// TIA Portal V17 export
// export: Created 2025-05-22T12:26:37.545947Z, ExportSetting WithDefaults, DisplayName Totally Integrated Automation Portal, DisplayVersion V17 Update 8, DisplayName TIA Portal Openness, DisplayVersion V17 Update 8, DisplayName TIA Portal Version Control Interface, DisplayVersion V17, DisplayName SINAMICS Startdrive Advanced, DisplayVersion V17 SP2, DisplayName SINAMICS Startdrive G110M, G120, G120C, G120D, G120P, G115D, DisplayVersion V17 SP2, DisplayName SINAMICS Startdrive G130, G150, S120, S150, SINAMICS MV, S210, DisplayVersion V17 SP2, DisplayName STEP 7 Professional, DisplayVersion V17 Update 8, DisplayName SINUMERIK ONE STEP 7 Toolbox, DisplayVersion V17 Update 12, DisplayName SINUMERIK ONE PLC Basic Program Plus, DisplayVersion V17 Update 12, DisplayName SINUMERIK 840D sl STEP 7 Toolbox, DisplayVersion V17 Update 12, DisplayName STEP 7 Safety, DisplayVersion V17 Update 6, DisplayName WinCC Advanced, DisplayVersion V17 Update 8
FUNCTION_BLOCK "FB1502_PROTECTION_GAS_VALVE"   // FB1502, LAD
{ S7_Optimized_Access := 'FALSE' }
VERSION : 0.1
// stored: AutoNumber false, IsIECCheckEnabled false, SetENOAutomatically false, UDAEnableTagReadback false
   VAR_INPUT
      FLOW_INPUT : Real;   // FLOW INPUT
      TEMPERATURE_INPUT : Real;   // TEMPERATURE INPUT
      LASER_READY_INPUT : Bool;   // LASER READY INPUT
      SWITCH_ON_CONDITIONS : Bool;   // SWITCH ON CONDITIONS
      SWITCH_OFF_CONDITIONS : Bool;   // SWITCH OFF CONDITIONS
      HMI_LINE_REQUEST : Bool;   // HMI LINE REQUEST
      SWITCH_ON_AUTO_REQUEST : Bool;   // AUTO SWITCH ON REQUEST
      SWITCH_OFF_AUTO_REQUEST : Bool;   // AUTO SWITCH OFF REQUEST
      SWITCH_OFF_GLOBAL_REQUEST : Bool;   // SWITCH OFF GLOBAL REQUEST (AUTO/SEMI/MAN)
      POWDER_ENABLED : Bool;
      UNIT_ALARM : UInt;   // UNIT NUMBER MIN. NUMBER=1 MAX. NUMBER=4
      STATION_ALARM : UInt;   // STATION NUMBER MIN. NUMBER=0 MAX. NUMBER=4
   END_VAR
   VAR_OUTPUT
      SWITCHED_ON : Bool;   // SWITCHED ON
      SWITCHED_OFF : Bool;   // SWITCHED OFF
      SIMULTANEITY_ALARM : Bool;   // SIMULTANEITY ALARM
      TIME_EXCEEDED_ALARM : Bool;   // TIME EXCEEDED ALARM
      SWITCH_ON_ALARM : Bool;   // SWITCH ON ALARM
      SWITCH_OFF_ALARM : Bool;   // SWITCH OFF ALARM
      GAS_FLOW_LOW_WARNING : Bool;   // GAS FLOW LOW WARNING
      GAS_FLOW_LOW_ALARM : Bool;   // GAS FLOW LOW ALARM
      GAS_FLOW_HIGH_WARNING : Bool;   // GAS FLOW HIGH WARNING
      GAS_FLOW_HIGH_ALARM : Bool;   // GAS FLOW HIGH ALARM
      GAS_TEMP_LOW_WARNING : Bool;   // GAS TEMPERATURE LOW WARNING
      GAS_TEMP_LOW_ALARM : Bool;   // GAS TEMPERATURE LOW ALARM
      GAS_TEMP_HIGH_WARNING : Bool;   // GAS TEMPERATURE HIGH WARNING
      GAS_TEMP_HIGH_ALARM : Bool;   // GAS TEMPERATURE HIGH ALARM
      ANY_ALARM_PRESENT : Bool;   // ANY ALARM PRESENT
      HMI_MOTION_EXECUTABILITY_LEFT : Bool;   // HMI MOTION EXECUTABILITY LEFT
      HMI_MOTION_EXECUTABILITY_RIGHT : Bool;   // HMI MOTION EXECUTABILITY RIGHT
      HMI_MOTION_END_POS_LEFT : Bool;   // HMI MOTION END POSITION LEFT
      HMI_MOTION_END_POS_RIGHT : Bool;   // HMI MOTION END POSITION RIGHT
      HMI_MOTION_ACTIVE_LEFT : Bool;   // HMI MOTION ACTIVE LEFT
      HMI_MOTION_ACTIVE_RIGHT : Bool;   // HMI MOTION ACTIVE RIGHT
      GAS_FLOW_SETPOINT : Real;   // GAS FLOW SETPOINT
      SWITCH_ON : Bool;   // SWITCH ON OUTPUT
      SWITCH_OFF : Bool;   // SWITCH OFF OUTPUT
   END_VAR
   VAR DB_SPECIFIC
      VALVE { S7_SetPoint := 'True'} : "ASPIRATION";
      HMI_VARIBLES : Struct
         HMI_GAS_FLOW_SETPOINT { S7_SetPoint := 'True'} : Real;
         GAS_FLOW_LOW_WARNING_VALUE : Real;
         GAS_FLOW_LOW_ALARM_VALUE : Real;
         GAS_FLOW_HIGH_WARNING_VALUE : Real;
         GAS_FLOW_HIGH_ALARM_VALUE : Real;
         TEMP_LOW_WARNING_VALUE : Real;
         TEMP_LOW_ALARM_VALUE : Real;
         TEMP_HIGH_WARNING_VALUE : Real;
         TEMP_HIGH_ALARM_VALUE : Real;
      END_STRUCT;
      FLOW_VALUE : Real;
      AUX_TEMP { S7_SetPoint := 'True'} : Real;   // AUX TEMPERATURE
      TEMPERATURE_VALUE { S7_SetPoint := 'True'} : Real;   // TEMPERATURE VALUE
      TIMER_SWITCHED_ON { S7_SetPoint := 'True'} : TON_TIME;   // SWITCHED ON TIMER
      TIMER_SWITCHED_OFF { S7_SetPoint := 'True'} : TON_TIME;   // SWITCHED OFF TIMER
      TIMER_SIMULTANEITY { S7_SetPoint := 'True'} : TON_TIME;   // SIMULTANEITY TIMER
      TIMER_TIME_EXCEEDED { S7_SetPoint := 'True'} : TON_TIME;   // TIME EXCEEDED TIMER
      GAS_FLOW_LOW_WARNING_DELAY { S7_SetPoint := 'True'} : TON_TIME;
      GAS_FLOW_LOW_ALARM_DELAY { S7_SetPoint := 'True'} : TON_TIME;
      PULSE { S7_SetPoint := 'True'} : Bool;
   END_VAR
   VAR_TEMP
      DB_NUMBER : DInt;   // DB NUMBER FOR ALARM AND HELP DECODING
   END_VAR
   // TIMER_SWITCHED_ON.PT := T#100MS;
   // TIMER_SWITCHED_OFF.PT := T#300MS;
   // TIMER_SIMULTANEITY.PT := T#100MS;
   // TIMER_TIME_EXCEEDED.PT := T#2S;
   VAR_TEMP   // added for the SCL form of the ladder/FBD networks
      _w1 : Bool;
      _w2 : Bool;
   END_VAR
BEGIN

NETWORK
TITLE = READ INSTANCE DB
      L     DINO;
      +     10#800000;
      T     #DB_NUMBER;


REGION Network 2: INPUT
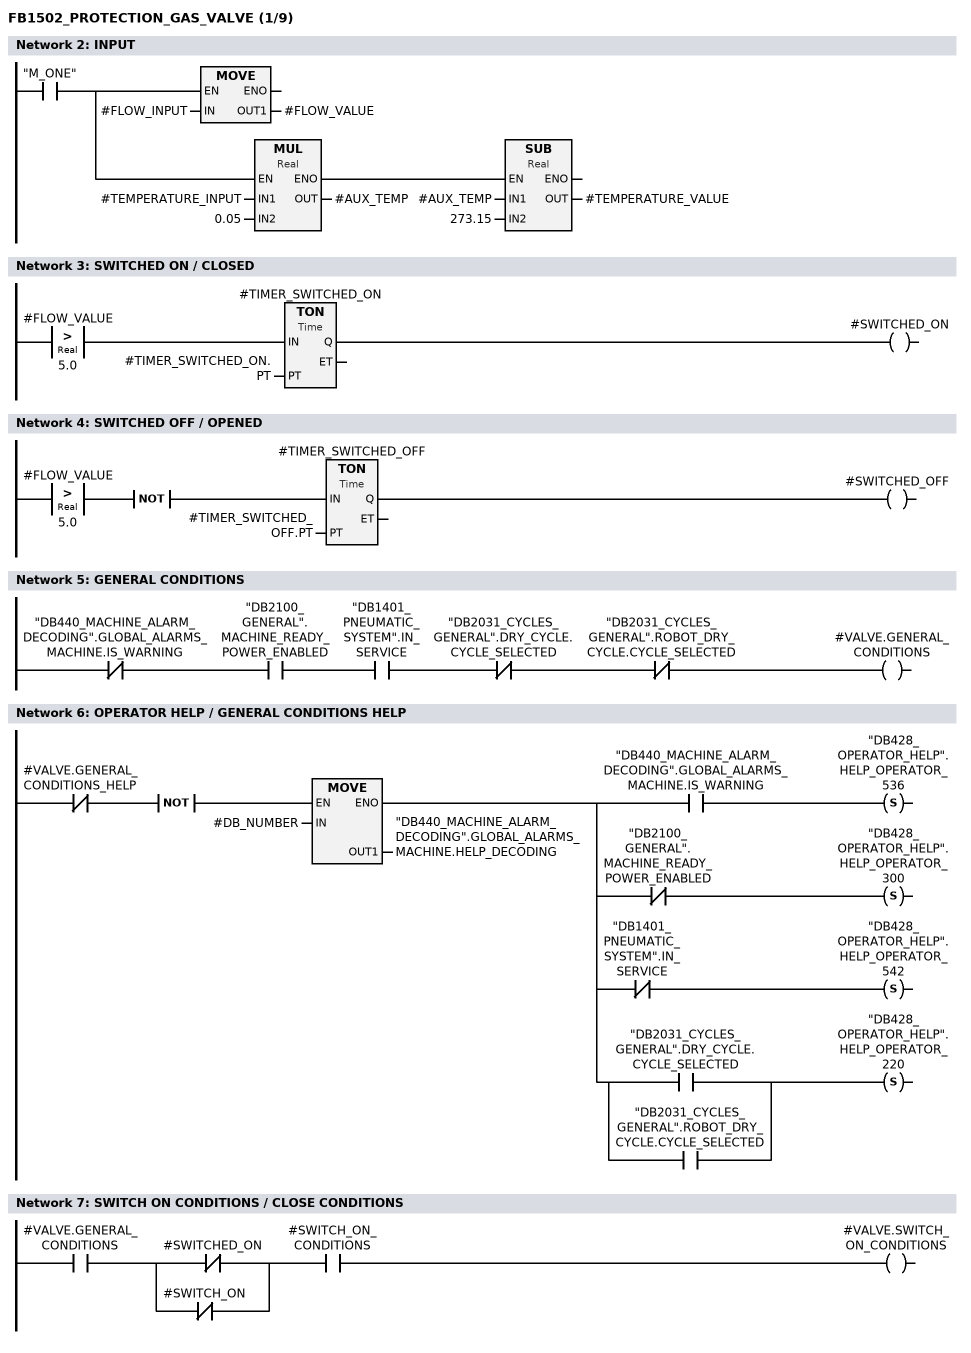
   RUNG wire#powerrail
      Contact( "M_ONE" )
      wire#w1
      Move(in := #FLOW_INPUT, out1 => #FLOW_VALUE)
   END_RUNG
   RUNG wire#w1
      { S7_Templates := "SrcType := Real" } Mul(in1 := #TEMPERATURE_INPUT, in2 := 0.05, out => #AUX_TEMP)
      { S7_Templates := "SrcType := Real" } Sub(in1 := #AUX_TEMP, in2 := 273.15, out => #TEMPERATURE_VALUE)
   END_RUNG
   // the same network as SCL:
   IF "M_ONE" THEN
       #FLOW_VALUE := #FLOW_INPUT;
       #AUX_TEMP := #TEMPERATURE_INPUT * 0.05;
       #TEMPERATURE_VALUE := #AUX_TEMP - 273.15;
   END_IF;
END_REGION

REGION Network 3: SWITCHED ON / CLOSED
   RUNG wire#powerrail
      { S7_Templates := "SrcType := Real" } GT_Contact(in1 := #FLOW_VALUE, in2 := 5.0)
      { S7_Templates := "time_type := Time" } #TIMER_SWITCHED_ON.TON(pt := #TIMER_SWITCHED_ON.PT, et =>)
      Coil( #SWITCHED_ON )
   END_RUNG
   // the same network as SCL:
   #TIMER_SWITCHED_ON(IN := #FLOW_VALUE > 5.0, PT := #TIMER_SWITCHED_ON.PT);   // TON
   #SWITCHED_ON := #TIMER_SWITCHED_ON.Q;
END_REGION

REGION Network 4: SWITCHED OFF / OPENED
   RUNG wire#powerrail
      { S7_Templates := "SrcType := Real" } GT_Contact(in1 := #FLOW_VALUE, in2 := 5.0)
      Not()
      { S7_Templates := "time_type := Time" } #TIMER_SWITCHED_OFF.TON(pt := #TIMER_SWITCHED_OFF.PT, et =>)
      Coil( #SWITCHED_OFF )
   END_RUNG
   // the same network as SCL:
   #TIMER_SWITCHED_OFF(IN := NOT (#FLOW_VALUE > 5.0), PT := #TIMER_SWITCHED_OFF.PT);   // TON
   #SWITCHED_OFF := #TIMER_SWITCHED_OFF.Q;
END_REGION

REGION Network 5: GENERAL CONDITIONS
   RUNG wire#powerrail
      I_Contact( "DB440_MACHINE_ALARM_DECODING".GLOBAL_ALARMS_MACHINE.IS_WARNING )
      Contact( "DB2100_GENERAL".MACHINE_READY_POWER_ENABLED )
      Contact( "DB1401_PNEUMATIC_SYSTEM".IN_SERVICE )
      I_Contact( "DB2031_CYCLES_GENERAL".DRY_CYCLE.CYCLE_SELECTED )
      I_Contact( "DB2031_CYCLES_GENERAL".ROBOT_DRY_CYCLE.CYCLE_SELECTED )
      Coil( #VALVE.GENERAL_CONDITIONS )
   END_RUNG
   // the same network as SCL:
   #VALVE.GENERAL_CONDITIONS := NOT "DB440_MACHINE_ALARM_DECODING".GLOBAL_ALARMS_MACHINE.IS_WARNING AND "DB2100_GENERAL".MACHINE_READY_POWER_ENABLED AND "DB1401_PNEUMATIC_SYSTEM".IN_SERVICE AND NOT "DB2031_CYCLES_GENERAL".DRY_CYCLE.CYCLE_SELECTED AND NOT "DB2031_CYCLES_GENERAL".ROBOT_DRY_CYCLE.CYCLE_SELECTED;
END_REGION

REGION Network 6: OPERATOR HELP / GENERAL CONDITIONS HELP
   RUNG wire#powerrail
      I_Contact( #VALVE.GENERAL_CONDITIONS_HELP )
      Not()
      { S7_GenerateENO := "TRUE" } Move(in := #DB_NUMBER, out1 => "DB440_MACHINE_ALARM_DECODING".GLOBAL_ALARMS_MACHINE.HELP_DECODING)
      wire#w1
      Contact( "DB440_MACHINE_ALARM_DECODING".GLOBAL_ALARMS_MACHINE.IS_WARNING )
      S_Coil( "DB428_OPERATOR_HELP".HELP_OPERATOR_536 )
   END_RUNG
   RUNG wire#w1
      I_Contact( "DB2100_GENERAL".MACHINE_READY_POWER_ENABLED )
      S_Coil( "DB428_OPERATOR_HELP".HELP_OPERATOR_300 )
   END_RUNG
   RUNG wire#w1
      I_Contact( "DB1401_PNEUMATIC_SYSTEM".IN_SERVICE )
      S_Coil( "DB428_OPERATOR_HELP".HELP_OPERATOR_542 )
   END_RUNG
   RUNG wire#w1
      Contact( "DB2031_CYCLES_GENERAL".DRY_CYCLE.CYCLE_SELECTED )
      wire#w2
      S_Coil( "DB428_OPERATOR_HELP".HELP_OPERATOR_220 )
   END_RUNG
   RUNG wire#w1
      Contact( "DB2031_CYCLES_GENERAL".ROBOT_DRY_CYCLE.CYCLE_SELECTED )
   END_RUNG wire#w2
   // the same network as SCL:
   // ENO of a box is taken as its EN; it also drops when the box reports an error
   #_w1 := NOT (NOT #VALVE.GENERAL_CONDITIONS_HELP);
   IF #_w1 THEN "DB440_MACHINE_ALARM_DECODING".GLOBAL_ALARMS_MACHINE.HELP_DECODING := #DB_NUMBER; END_IF;
   IF #_w1 AND "DB440_MACHINE_ALARM_DECODING".GLOBAL_ALARMS_MACHINE.IS_WARNING THEN
       "DB428_OPERATOR_HELP".HELP_OPERATOR_536 := TRUE;
   END_IF;
   IF #_w1 AND NOT "DB2100_GENERAL".MACHINE_READY_POWER_ENABLED THEN
       "DB428_OPERATOR_HELP".HELP_OPERATOR_300 := TRUE;
   END_IF;
   IF #_w1 AND NOT "DB1401_PNEUMATIC_SYSTEM".IN_SERVICE THEN
       "DB428_OPERATOR_HELP".HELP_OPERATOR_542 := TRUE;
   END_IF;
   IF #_w1 AND ("DB2031_CYCLES_GENERAL".DRY_CYCLE.CYCLE_SELECTED OR "DB2031_CYCLES_GENERAL".ROBOT_DRY_CYCLE.CYCLE_SELECTED) THEN
       "DB428_OPERATOR_HELP".HELP_OPERATOR_220 := TRUE;
   END_IF;
END_REGION

REGION Network 7: SWITCH ON CONDITIONS / CLOSE CONDITIONS
   RUNG wire#powerrail
      Contact( #VALVE.GENERAL_CONDITIONS )
      wire#w1
      I_Contact( #SWITCHED_ON )
      wire#w2
      Contact( #SWITCH_ON_CONDITIONS )
      Coil( #VALVE.SWITCH_ON_CONDITIONS )
   END_RUNG
   RUNG wire#w1
      I_Contact( #SWITCH_ON )
   END_RUNG wire#w2
   // the same network as SCL:
   #VALVE.SWITCH_ON_CONDITIONS := #VALVE.GENERAL_CONDITIONS AND (NOT #SWITCHED_ON OR NOT #SWITCH_ON) AND #SWITCH_ON_CONDITIONS;
END_REGION

REGION Network 8: OPERATOR HELP / CLOSE CONDITIONS HELP
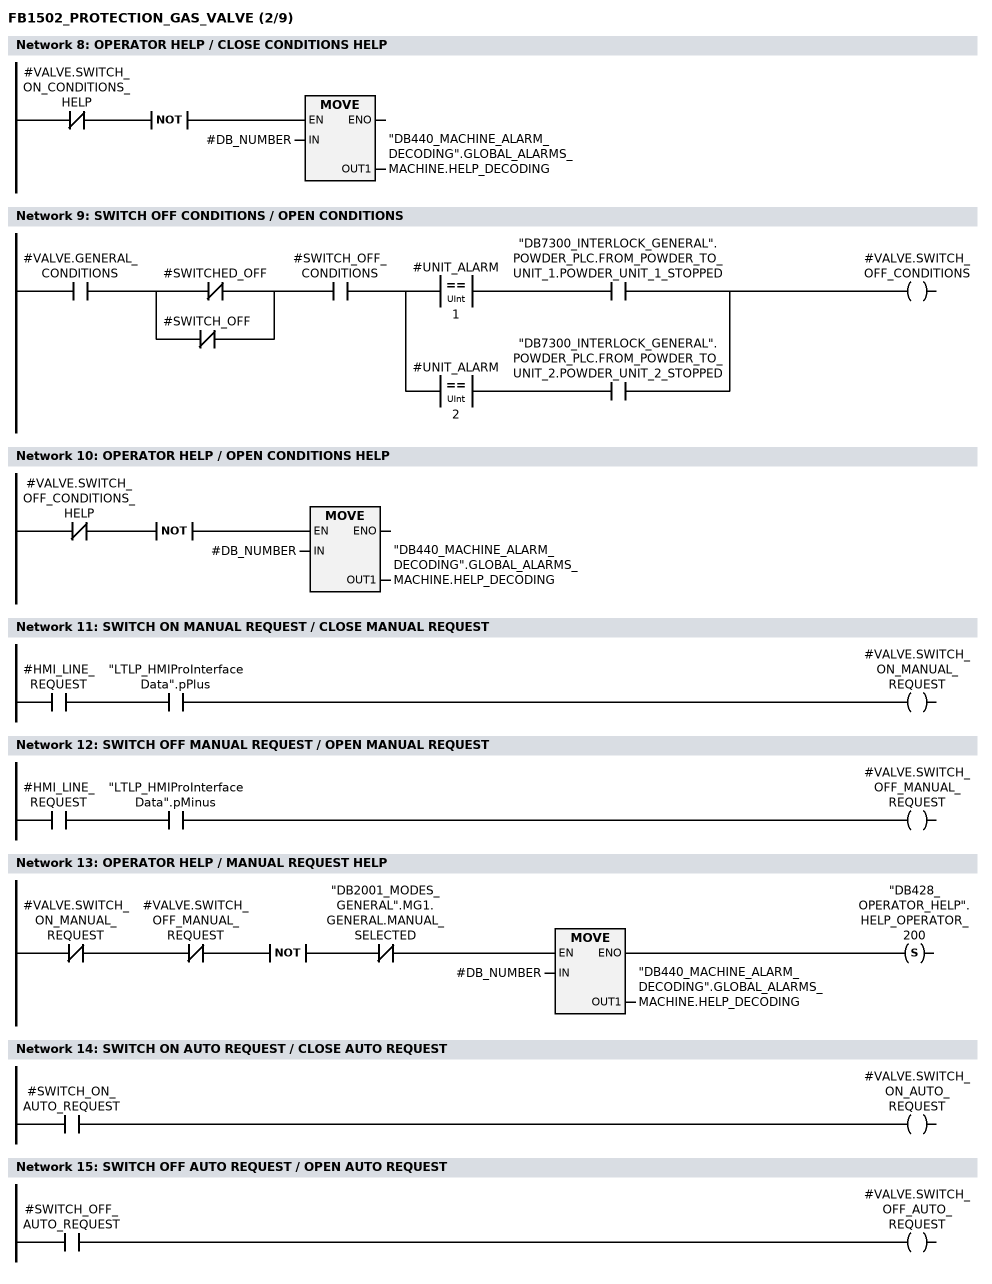
   RUNG wire#powerrail
      I_Contact( #VALVE.SWITCH_ON_CONDITIONS_HELP )
      Not()
      { S7_GenerateENO := "TRUE" } Move(in := #DB_NUMBER, out1 => "DB440_MACHINE_ALARM_DECODING".GLOBAL_ALARMS_MACHINE.HELP_DECODING)
   END_RUNG
   // the same network as SCL:
   IF NOT (NOT #VALVE.SWITCH_ON_CONDITIONS_HELP) THEN
       "DB440_MACHINE_ALARM_DECODING".GLOBAL_ALARMS_MACHINE.HELP_DECODING := #DB_NUMBER;
   END_IF;
END_REGION

REGION Network 9: SWITCH OFF CONDITIONS / OPEN CONDITIONS
   RUNG wire#powerrail
      Contact( #VALVE.GENERAL_CONDITIONS )
      wire#w1
      I_Contact( #SWITCHED_OFF )
      wire#w2
      Contact( #SWITCH_OFF_CONDITIONS )
      wire#w3
      { S7_Templates := "SrcType := UInt" } EQ_Contact(in1 := #UNIT_ALARM, in2 := 1)
      Contact( "DB7300_INTERLOCK_GENERAL".POWDER_PLC.FROM_POWDER_TO_UNIT_1.POWDER_UNIT_1_STOPPED )
      wire#w4
      Coil( #VALVE.SWITCH_OFF_CONDITIONS )
   END_RUNG
   RUNG wire#w1
      I_Contact( #SWITCH_OFF )
   END_RUNG wire#w2
   RUNG wire#w3
      { S7_Templates := "SrcType := UInt" } EQ_Contact(in1 := #UNIT_ALARM, in2 := 2)
      Contact( "DB7300_INTERLOCK_GENERAL".POWDER_PLC.FROM_POWDER_TO_UNIT_2.POWDER_UNIT_2_STOPPED )
   END_RUNG wire#w4
   // the same network as SCL:
   #VALVE.SWITCH_OFF_CONDITIONS := #VALVE.GENERAL_CONDITIONS AND (NOT #SWITCHED_OFF OR NOT #SWITCH_OFF) AND #SWITCH_OFF_CONDITIONS AND (((#UNIT_ALARM = 1) AND "DB7300_INTERLOCK_GENERAL".POWDER_PLC.FROM_POWDER_TO_UNIT_1.POWDER_UNIT_1_STOPPED) OR ((#UNIT_ALARM = 2) AND "DB7300_INTERLOCK_GENERAL".POWDER_PLC.FROM_POWDER_TO_UNIT_2.POWDER_UNIT_2_STOPPED));
END_REGION

REGION Network 10: OPERATOR HELP / OPEN CONDITIONS HELP
   RUNG wire#powerrail
      I_Contact( #VALVE.SWITCH_OFF_CONDITIONS_HELP )
      Not()
      { S7_GenerateENO := "TRUE" } Move(in := #DB_NUMBER, out1 => "DB440_MACHINE_ALARM_DECODING".GLOBAL_ALARMS_MACHINE.HELP_DECODING)
   END_RUNG
   // the same network as SCL:
   IF NOT (NOT #VALVE.SWITCH_OFF_CONDITIONS_HELP) THEN
       "DB440_MACHINE_ALARM_DECODING".GLOBAL_ALARMS_MACHINE.HELP_DECODING := #DB_NUMBER;
   END_IF;
END_REGION

REGION Network 11: SWITCH ON MANUAL REQUEST / CLOSE MANUAL REQUEST
   RUNG wire#powerrail
      Contact( #HMI_LINE_REQUEST )
      Contact( "LTLP_HMIProInterfaceData".pPlus )
      Coil( #VALVE.SWITCH_ON_MANUAL_REQUEST )
   END_RUNG
   // the same network as SCL:
   #VALVE.SWITCH_ON_MANUAL_REQUEST := #HMI_LINE_REQUEST AND "LTLP_HMIProInterfaceData".pPlus;
END_REGION

REGION Network 12: SWITCH OFF MANUAL REQUEST / OPEN MANUAL REQUEST
   RUNG wire#powerrail
      Contact( #HMI_LINE_REQUEST )
      Contact( "LTLP_HMIProInterfaceData".pMinus )
      Coil( #VALVE.SWITCH_OFF_MANUAL_REQUEST )
   END_RUNG
   // the same network as SCL:
   #VALVE.SWITCH_OFF_MANUAL_REQUEST := #HMI_LINE_REQUEST AND "LTLP_HMIProInterfaceData".pMinus;
END_REGION

REGION Network 13: OPERATOR HELP / MANUAL REQUEST HELP
   RUNG wire#powerrail
      I_Contact( #VALVE.SWITCH_ON_MANUAL_REQUEST )
      I_Contact( #VALVE.SWITCH_OFF_MANUAL_REQUEST )
      Not()
      I_Contact( "DB2001_MODES_GENERAL".MG1.GENERAL.MANUAL_SELECTED )
      { S7_GenerateENO := "TRUE" } Move(in := #DB_NUMBER, out1 => "DB440_MACHINE_ALARM_DECODING".GLOBAL_ALARMS_MACHINE.HELP_DECODING)
      S_Coil( "DB428_OPERATOR_HELP".HELP_OPERATOR_200 )
   END_RUNG
   // the same network as SCL:
   // ENO of a box is taken as its EN; it also drops when the box reports an error
   IF NOT (NOT #VALVE.SWITCH_ON_MANUAL_REQUEST AND NOT #VALVE.SWITCH_OFF_MANUAL_REQUEST) AND NOT "DB2001_MODES_GENERAL".MG1.GENERAL.MANUAL_SELECTED THEN
       "DB440_MACHINE_ALARM_DECODING".GLOBAL_ALARMS_MACHINE.HELP_DECODING := #DB_NUMBER;
       "DB428_OPERATOR_HELP".HELP_OPERATOR_200 := TRUE;
   END_IF;
END_REGION

REGION Network 14: SWITCH ON AUTO REQUEST / CLOSE AUTO REQUEST
   RUNG wire#powerrail
      Contact( #SWITCH_ON_AUTO_REQUEST )
      Coil( #VALVE.SWITCH_ON_AUTO_REQUEST )
   END_RUNG
   // the same network as SCL:
   #VALVE.SWITCH_ON_AUTO_REQUEST := #SWITCH_ON_AUTO_REQUEST;
END_REGION

REGION Network 15: SWITCH OFF AUTO REQUEST / OPEN AUTO REQUEST
   RUNG wire#powerrail
      Contact( #SWITCH_OFF_AUTO_REQUEST )
      Coil( #VALVE.SWITCH_OFF_AUTO_REQUEST )
   END_RUNG
   // the same network as SCL:
   #VALVE.SWITCH_OFF_AUTO_REQUEST := #SWITCH_OFF_AUTO_REQUEST;
END_REGION

REGION Network 16: SWITCH ON GLOBAL REQUEST / CLOSE GLOBAL REQUEST
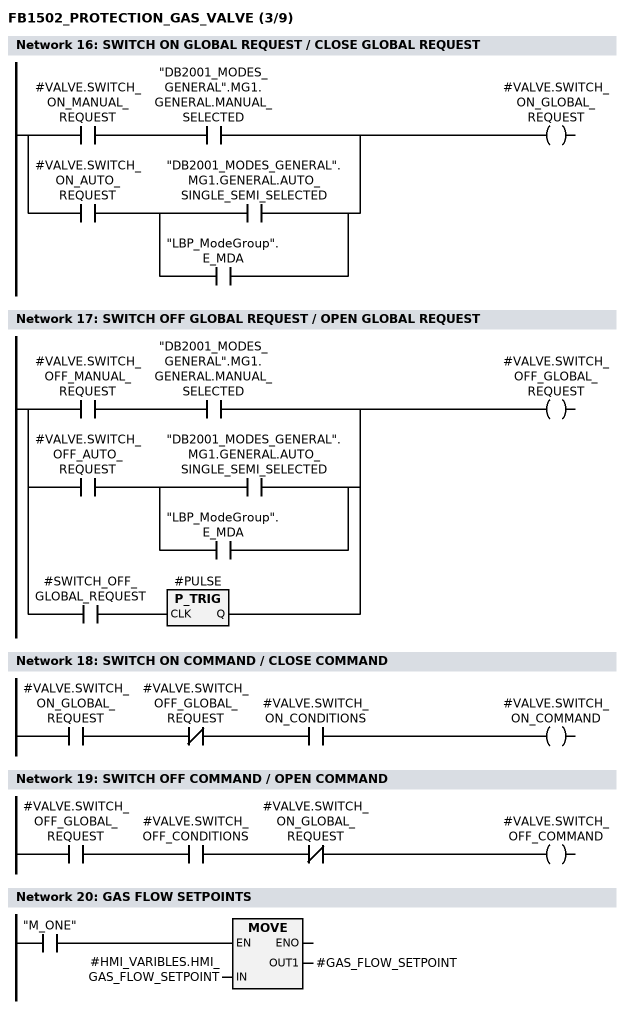
   RUNG wire#powerrail
      Contact( #VALVE.SWITCH_ON_MANUAL_REQUEST )
      Contact( "DB2001_MODES_GENERAL".MG1.GENERAL.MANUAL_SELECTED )
      wire#w1
      Coil( #VALVE.SWITCH_ON_GLOBAL_REQUEST )
   END_RUNG
   RUNG wire#powerrail
      Contact( #VALVE.SWITCH_ON_AUTO_REQUEST )
      wire#w2
      Contact( "DB2001_MODES_GENERAL".MG1.GENERAL.AUTO_SINGLE_SEMI_SELECTED )
   END_RUNG wire#w1
   RUNG wire#w2
      Contact( "LBP_ModeGroup".E_MDA )
   END_RUNG wire#w1
   // the same network as SCL:
   #VALVE.SWITCH_ON_GLOBAL_REQUEST := (#VALVE.SWITCH_ON_MANUAL_REQUEST AND "DB2001_MODES_GENERAL".MG1.GENERAL.MANUAL_SELECTED) OR (#VALVE.SWITCH_ON_AUTO_REQUEST AND ("DB2001_MODES_GENERAL".MG1.GENERAL.AUTO_SINGLE_SEMI_SELECTED OR "LBP_ModeGroup".E_MDA));
END_REGION

REGION Network 17: SWITCH OFF GLOBAL REQUEST / OPEN GLOBAL REQUEST
   RUNG wire#powerrail
      Contact( #VALVE.SWITCH_OFF_MANUAL_REQUEST )
      Contact( "DB2001_MODES_GENERAL".MG1.GENERAL.MANUAL_SELECTED )
      wire#w1
      Coil( #VALVE.SWITCH_OFF_GLOBAL_REQUEST )
   END_RUNG
   RUNG wire#powerrail
      Contact( #VALVE.SWITCH_OFF_AUTO_REQUEST )
      wire#w2
      Contact( "DB2001_MODES_GENERAL".MG1.GENERAL.AUTO_SINGLE_SEMI_SELECTED )
   END_RUNG wire#w1
   RUNG wire#w2
      Contact( "LBP_ModeGroup".E_MDA )
   END_RUNG wire#w1
   RUNG wire#powerrail
      Contact( #SWITCH_OFF_GLOBAL_REQUEST )
      P_Trig( #PULSE )
   END_RUNG wire#w1
   // the same network as SCL:
   #_w1 := #SWITCH_OFF_GLOBAL_REQUEST AND NOT #PULSE;   // rising edge
   #PULSE := #SWITCH_OFF_GLOBAL_REQUEST;
   #VALVE.SWITCH_OFF_GLOBAL_REQUEST := (#VALVE.SWITCH_OFF_MANUAL_REQUEST AND "DB2001_MODES_GENERAL".MG1.GENERAL.MANUAL_SELECTED) OR (#VALVE.SWITCH_OFF_AUTO_REQUEST AND ("DB2001_MODES_GENERAL".MG1.GENERAL.AUTO_SINGLE_SEMI_SELECTED OR "LBP_ModeGroup".E_MDA)) OR #_w1;
END_REGION

REGION Network 18: SWITCH ON COMMAND / CLOSE COMMAND
   RUNG wire#powerrail
      Contact( #VALVE.SWITCH_ON_GLOBAL_REQUEST )
      I_Contact( #VALVE.SWITCH_OFF_GLOBAL_REQUEST )
      Contact( #VALVE.SWITCH_ON_CONDITIONS )
      Coil( #VALVE.SWITCH_ON_COMMAND )
   END_RUNG
   // the same network as SCL:
   #VALVE.SWITCH_ON_COMMAND := #VALVE.SWITCH_ON_GLOBAL_REQUEST AND NOT #VALVE.SWITCH_OFF_GLOBAL_REQUEST AND #VALVE.SWITCH_ON_CONDITIONS;
END_REGION

REGION Network 19: SWITCH OFF COMMAND / OPEN COMMAND
   RUNG wire#powerrail
      Contact( #VALVE.SWITCH_OFF_GLOBAL_REQUEST )
      Contact( #VALVE.SWITCH_OFF_CONDITIONS )
      I_Contact( #VALVE.SWITCH_ON_GLOBAL_REQUEST )
      Coil( #VALVE.SWITCH_OFF_COMMAND )
   END_RUNG
   // the same network as SCL:
   #VALVE.SWITCH_OFF_COMMAND := #VALVE.SWITCH_OFF_GLOBAL_REQUEST AND #VALVE.SWITCH_OFF_CONDITIONS AND NOT #VALVE.SWITCH_ON_GLOBAL_REQUEST;
END_REGION

REGION Network 20: GAS FLOW SETPOINTS
   RUNG wire#powerrail
      Contact( "M_ONE" )
      Move(in := #HMI_VARIBLES.HMI_GAS_FLOW_SETPOINT, out1 => #GAS_FLOW_SETPOINT)
   END_RUNG
   // the same network as SCL:
   IF "M_ONE" THEN #GAS_FLOW_SETPOINT := #HMI_VARIBLES.HMI_GAS_FLOW_SETPOINT; END_IF;
END_REGION

REGION Network 21: SWITCH ON OUTPUT / CLOSE
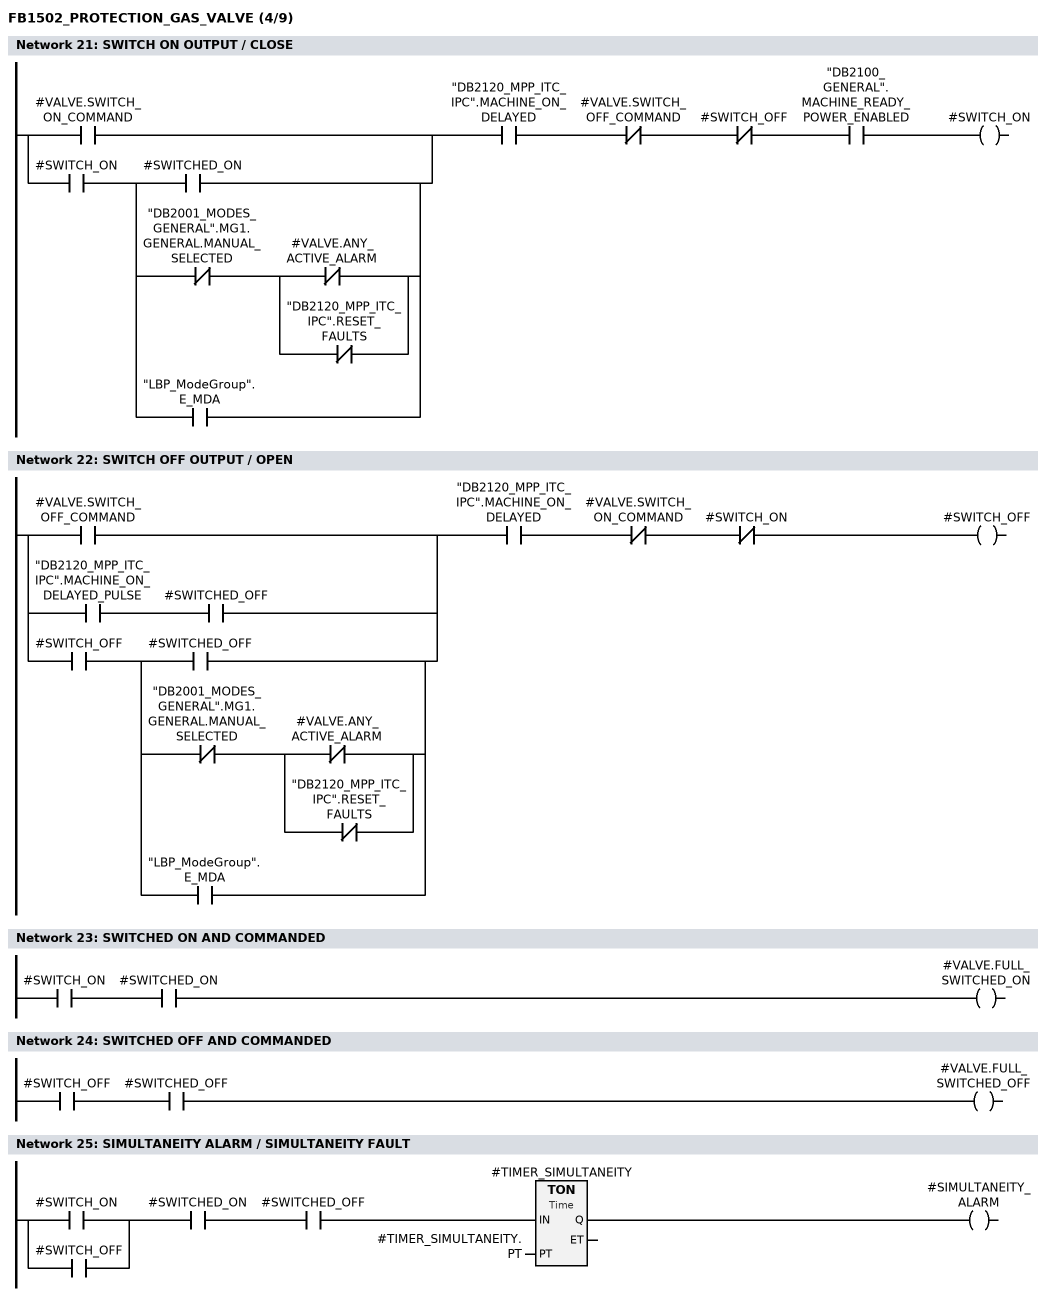
   RUNG wire#powerrail
      Contact( #VALVE.SWITCH_ON_COMMAND )
      wire#w1
      Contact( "DB2120_MPP_ITC_IPC".MACHINE_ON_DELAYED )
      I_Contact( #VALVE.SWITCH_OFF_COMMAND )
      I_Contact( #SWITCH_OFF )
      Contact( "DB2100_GENERAL".MACHINE_READY_POWER_ENABLED )
      Coil( #SWITCH_ON )
   END_RUNG
   RUNG wire#powerrail
      Contact( #SWITCH_ON )
      wire#w2
      Contact( #SWITCHED_ON )
   END_RUNG wire#w1
   RUNG wire#w2
      I_Contact( "DB2001_MODES_GENERAL".MG1.GENERAL.MANUAL_SELECTED )
      wire#w3
      I_Contact( #VALVE.ANY_ACTIVE_ALARM )
   END_RUNG wire#w1
   RUNG wire#w3
      I_Contact( "DB2120_MPP_ITC_IPC".RESET_FAULTS )
   END_RUNG wire#w1
   RUNG wire#w2
      Contact( "LBP_ModeGroup".E_MDA )
   END_RUNG wire#w1
   // the same network as SCL:
   #SWITCH_ON := (#VALVE.SWITCH_ON_COMMAND OR (#SWITCH_ON AND (#SWITCHED_ON OR (NOT "DB2001_MODES_GENERAL".MG1.GENERAL.MANUAL_SELECTED AND (NOT #VALVE.ANY_ACTIVE_ALARM OR NOT "DB2120_MPP_ITC_IPC".RESET_FAULTS)) OR "LBP_ModeGroup".E_MDA))) AND "DB2120_MPP_ITC_IPC".MACHINE_ON_DELAYED AND NOT #VALVE.SWITCH_OFF_COMMAND AND NOT #SWITCH_OFF AND "DB2100_GENERAL".MACHINE_READY_POWER_ENABLED;
END_REGION

REGION Network 22: SWITCH OFF OUTPUT / OPEN
   RUNG wire#powerrail
      Contact( #VALVE.SWITCH_OFF_COMMAND )
      wire#w1
      Contact( "DB2120_MPP_ITC_IPC".MACHINE_ON_DELAYED )
      I_Contact( #VALVE.SWITCH_ON_COMMAND )
      I_Contact( #SWITCH_ON )
      Coil( #SWITCH_OFF )
   END_RUNG
   RUNG wire#powerrail
      Contact( "DB2120_MPP_ITC_IPC".MACHINE_ON_DELAYED_PULSE )
      Contact( #SWITCHED_OFF )
   END_RUNG wire#w1
   RUNG wire#powerrail
      Contact( #SWITCH_OFF )
      wire#w2
      Contact( #SWITCHED_OFF )
   END_RUNG wire#w1
   RUNG wire#w2
      I_Contact( "DB2001_MODES_GENERAL".MG1.GENERAL.MANUAL_SELECTED )
      wire#w3
      I_Contact( #VALVE.ANY_ACTIVE_ALARM )
   END_RUNG wire#w1
   RUNG wire#w3
      I_Contact( "DB2120_MPP_ITC_IPC".RESET_FAULTS )
   END_RUNG wire#w1
   RUNG wire#w2
      Contact( "LBP_ModeGroup".E_MDA )
   END_RUNG wire#w1
   // the same network as SCL:
   #SWITCH_OFF := (#VALVE.SWITCH_OFF_COMMAND OR ("DB2120_MPP_ITC_IPC".MACHINE_ON_DELAYED_PULSE AND #SWITCHED_OFF) OR (#SWITCH_OFF AND (#SWITCHED_OFF OR (NOT "DB2001_MODES_GENERAL".MG1.GENERAL.MANUAL_SELECTED AND (NOT #VALVE.ANY_ACTIVE_ALARM OR NOT "DB2120_MPP_ITC_IPC".RESET_FAULTS)) OR "LBP_ModeGroup".E_MDA))) AND "DB2120_MPP_ITC_IPC".MACHINE_ON_DELAYED AND NOT #VALVE.SWITCH_ON_COMMAND AND NOT #SWITCH_ON;
END_REGION

REGION Network 23: SWITCHED ON AND COMMANDED
   RUNG wire#powerrail
      Contact( #SWITCH_ON )
      Contact( #SWITCHED_ON )
      Coil( #VALVE.FULL_SWITCHED_ON )
   END_RUNG
   // the same network as SCL:
   #VALVE.FULL_SWITCHED_ON := #SWITCH_ON AND #SWITCHED_ON;
END_REGION

REGION Network 24: SWITCHED OFF AND COMMANDED
   RUNG wire#powerrail
      Contact( #SWITCH_OFF )
      Contact( #SWITCHED_OFF )
      Coil( #VALVE.FULL_SWITCHED_OFF )
   END_RUNG
   // the same network as SCL:
   #VALVE.FULL_SWITCHED_OFF := #SWITCH_OFF AND #SWITCHED_OFF;
END_REGION

REGION Network 25: SIMULTANEITY ALARM / SIMULTANEITY FAULT
   RUNG wire#powerrail
      Contact( #SWITCH_ON )
      wire#w1
      Contact( #SWITCHED_ON )
      Contact( #SWITCHED_OFF )
      { S7_Templates := "time_type := Time" } #TIMER_SIMULTANEITY.TON(pt := #TIMER_SIMULTANEITY.PT, et =>)
      Coil( #SIMULTANEITY_ALARM )
   END_RUNG
   RUNG wire#powerrail
      Contact( #SWITCH_OFF )
   END_RUNG wire#w1
   // the same network as SCL:
   #TIMER_SIMULTANEITY(IN := (#SWITCH_ON OR #SWITCH_OFF) AND #SWITCHED_ON AND #SWITCHED_OFF,   // TON
                       PT := #TIMER_SIMULTANEITY.PT);
   #SIMULTANEITY_ALARM := #TIMER_SIMULTANEITY.Q;
END_REGION

REGION Network 26: TIME EXCEEDED ALARM / TIME EXCEEDED
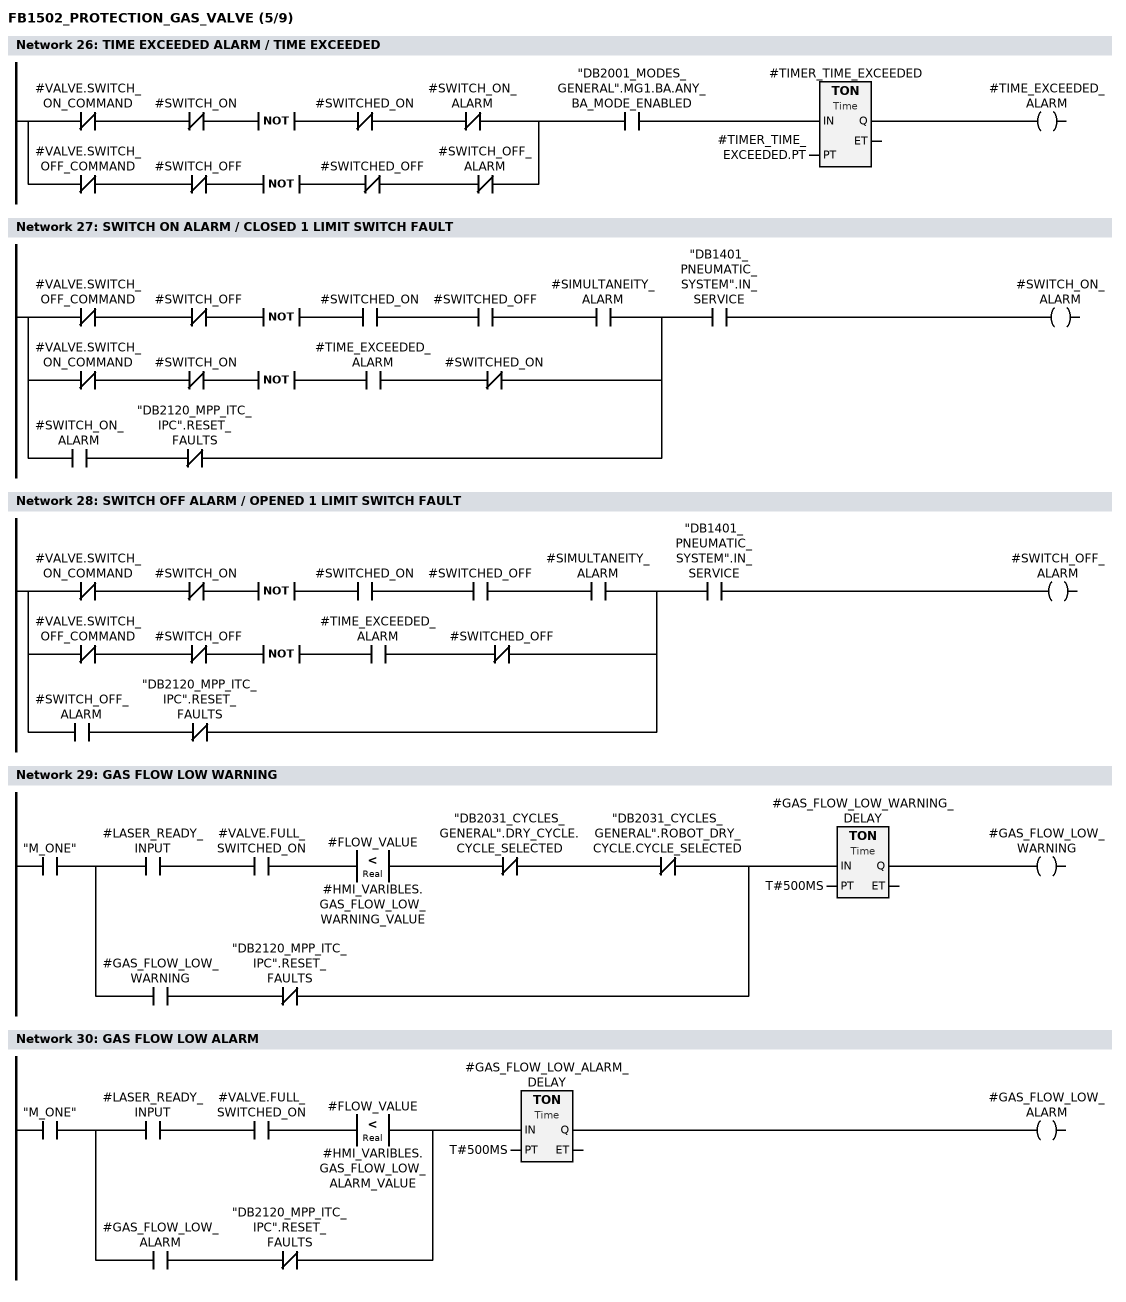
   RUNG wire#powerrail
      I_Contact( #VALVE.SWITCH_ON_COMMAND )
      I_Contact( #SWITCH_ON )
      Not()
      I_Contact( #SWITCHED_ON )
      I_Contact( #SWITCH_ON_ALARM )
      wire#w1
      Contact( "DB2001_MODES_GENERAL".MG1.BA.ANY_BA_MODE_ENABLED )
      { S7_Templates := "time_type := Time" } #TIMER_TIME_EXCEEDED.TON(pt := #TIMER_TIME_EXCEEDED.PT, et =>)
      Coil( #TIME_EXCEEDED_ALARM )
   END_RUNG
   RUNG wire#powerrail
      I_Contact( #VALVE.SWITCH_OFF_COMMAND )
      I_Contact( #SWITCH_OFF )
      Not()
      I_Contact( #SWITCHED_OFF )
      I_Contact( #SWITCH_OFF_ALARM )
   END_RUNG wire#w1
   // the same network as SCL:
   #TIMER_TIME_EXCEEDED(IN := ((NOT (NOT #VALVE.SWITCH_ON_COMMAND AND NOT #SWITCH_ON) AND NOT #SWITCHED_ON AND NOT #SWITCH_ON_ALARM) OR (NOT (NOT #VALVE.SWITCH_OFF_COMMAND AND NOT #SWITCH_OFF) AND NOT #SWITCHED_OFF AND NOT #SWITCH_OFF_ALARM)) AND "DB2001_MODES_GENERAL".MG1.BA.ANY_BA_MODE_ENABLED,   // TON
                        PT := #TIMER_TIME_EXCEEDED.PT);
   #TIME_EXCEEDED_ALARM := #TIMER_TIME_EXCEEDED.Q;
END_REGION

REGION Network 27: SWITCH ON ALARM / CLOSED 1 LIMIT SWITCH FAULT
   RUNG wire#powerrail
      I_Contact( #VALVE.SWITCH_OFF_COMMAND )
      I_Contact( #SWITCH_OFF )
      Not()
      Contact( #SWITCHED_ON )
      Contact( #SWITCHED_OFF )
      Contact( #SIMULTANEITY_ALARM )
      wire#w1
      Contact( "DB1401_PNEUMATIC_SYSTEM".IN_SERVICE )
      Coil( #SWITCH_ON_ALARM )
   END_RUNG
   RUNG wire#powerrail
      I_Contact( #VALVE.SWITCH_ON_COMMAND )
      I_Contact( #SWITCH_ON )
      Not()
      Contact( #TIME_EXCEEDED_ALARM )
      I_Contact( #SWITCHED_ON )
   END_RUNG wire#w1
   RUNG wire#powerrail
      Contact( #SWITCH_ON_ALARM )
      I_Contact( "DB2120_MPP_ITC_IPC".RESET_FAULTS )
   END_RUNG wire#w1
   // the same network as SCL:
   #SWITCH_ON_ALARM := ((NOT (NOT #VALVE.SWITCH_OFF_COMMAND AND NOT #SWITCH_OFF) AND #SWITCHED_ON AND #SWITCHED_OFF AND #SIMULTANEITY_ALARM) OR (NOT (NOT #VALVE.SWITCH_ON_COMMAND AND NOT #SWITCH_ON) AND #TIME_EXCEEDED_ALARM AND NOT #SWITCHED_ON) OR (#SWITCH_ON_ALARM AND NOT "DB2120_MPP_ITC_IPC".RESET_FAULTS)) AND "DB1401_PNEUMATIC_SYSTEM".IN_SERVICE;
END_REGION

REGION Network 28: SWITCH OFF ALARM / OPENED 1 LIMIT SWITCH FAULT
   RUNG wire#powerrail
      I_Contact( #VALVE.SWITCH_ON_COMMAND )
      I_Contact( #SWITCH_ON )
      Not()
      Contact( #SWITCHED_ON )
      Contact( #SWITCHED_OFF )
      Contact( #SIMULTANEITY_ALARM )
      wire#w1
      Contact( "DB1401_PNEUMATIC_SYSTEM".IN_SERVICE )
      Coil( #SWITCH_OFF_ALARM )
   END_RUNG
   RUNG wire#powerrail
      I_Contact( #VALVE.SWITCH_OFF_COMMAND )
      I_Contact( #SWITCH_OFF )
      Not()
      Contact( #TIME_EXCEEDED_ALARM )
      I_Contact( #SWITCHED_OFF )
   END_RUNG wire#w1
   RUNG wire#powerrail
      Contact( #SWITCH_OFF_ALARM )
      I_Contact( "DB2120_MPP_ITC_IPC".RESET_FAULTS )
   END_RUNG wire#w1
   // the same network as SCL:
   #SWITCH_OFF_ALARM := ((NOT (NOT #VALVE.SWITCH_ON_COMMAND AND NOT #SWITCH_ON) AND #SWITCHED_ON AND #SWITCHED_OFF AND #SIMULTANEITY_ALARM) OR (NOT (NOT #VALVE.SWITCH_OFF_COMMAND AND NOT #SWITCH_OFF) AND #TIME_EXCEEDED_ALARM AND NOT #SWITCHED_OFF) OR (#SWITCH_OFF_ALARM AND NOT "DB2120_MPP_ITC_IPC".RESET_FAULTS)) AND "DB1401_PNEUMATIC_SYSTEM".IN_SERVICE;
END_REGION

REGION Network 29: GAS FLOW LOW WARNING
   RUNG wire#powerrail
      Contact( "M_ONE" )
      wire#w1
      Contact( #LASER_READY_INPUT )
      Contact( #VALVE.FULL_SWITCHED_ON )
      { S7_Templates := "SrcType := Real" } LT_Contact(in1 := #FLOW_VALUE, in2 := #HMI_VARIBLES.GAS_FLOW_LOW_WARNING_VALUE)
      I_Contact( "DB2031_CYCLES_GENERAL".DRY_CYCLE.CYCLE_SELECTED )
      I_Contact( "DB2031_CYCLES_GENERAL".ROBOT_DRY_CYCLE.CYCLE_SELECTED )
      wire#w2
      { S7_Templates := "time_type := Time" } #GAS_FLOW_LOW_WARNING_DELAY.TON(pt := T#500MS, et =>)
      Coil( #GAS_FLOW_LOW_WARNING )
   END_RUNG
   RUNG wire#w1
      Contact( #GAS_FLOW_LOW_WARNING )
      I_Contact( "DB2120_MPP_ITC_IPC".RESET_FAULTS )
   END_RUNG wire#w2
   // the same network as SCL:
   #GAS_FLOW_LOW_WARNING_DELAY(IN := "M_ONE" AND ((#LASER_READY_INPUT AND #VALVE.FULL_SWITCHED_ON AND (#FLOW_VALUE < #HMI_VARIBLES.GAS_FLOW_LOW_WARNING_VALUE) AND NOT "DB2031_CYCLES_GENERAL".DRY_CYCLE.CYCLE_SELECTED AND NOT "DB2031_CYCLES_GENERAL".ROBOT_DRY_CYCLE.CYCLE_SELECTED) OR (#GAS_FLOW_LOW_WARNING AND NOT "DB2120_MPP_ITC_IPC".RESET_FAULTS)),   // TON
                           PT := T#500MS);
   #GAS_FLOW_LOW_WARNING := #GAS_FLOW_LOW_WARNING_DELAY.Q;
END_REGION

REGION Network 30: GAS FLOW LOW ALARM
   RUNG wire#powerrail
      Contact( "M_ONE" )
      wire#w1
      Contact( #LASER_READY_INPUT )
      Contact( #VALVE.FULL_SWITCHED_ON )
      { S7_Templates := "SrcType := Real" } LT_Contact(in1 := #FLOW_VALUE, in2 := #HMI_VARIBLES.GAS_FLOW_LOW_ALARM_VALUE)
      wire#w2
      { S7_Templates := "time_type := Time" } #GAS_FLOW_LOW_ALARM_DELAY.TON(pt := T#500MS, et =>)
      Coil( #GAS_FLOW_LOW_ALARM )
   END_RUNG
   RUNG wire#w1
      Contact( #GAS_FLOW_LOW_ALARM )
      I_Contact( "DB2120_MPP_ITC_IPC".RESET_FAULTS )
   END_RUNG wire#w2
   // the same network as SCL:
   #GAS_FLOW_LOW_ALARM_DELAY(IN := "M_ONE" AND ((#LASER_READY_INPUT AND #VALVE.FULL_SWITCHED_ON AND (#FLOW_VALUE < #HMI_VARIBLES.GAS_FLOW_LOW_ALARM_VALUE)) OR (#GAS_FLOW_LOW_ALARM AND NOT "DB2120_MPP_ITC_IPC".RESET_FAULTS)),   // TON
                           PT := T#500MS);
   #GAS_FLOW_LOW_ALARM := #GAS_FLOW_LOW_ALARM_DELAY.Q;
END_REGION

REGION Network 31: GAS FLOW HIGH WARNING
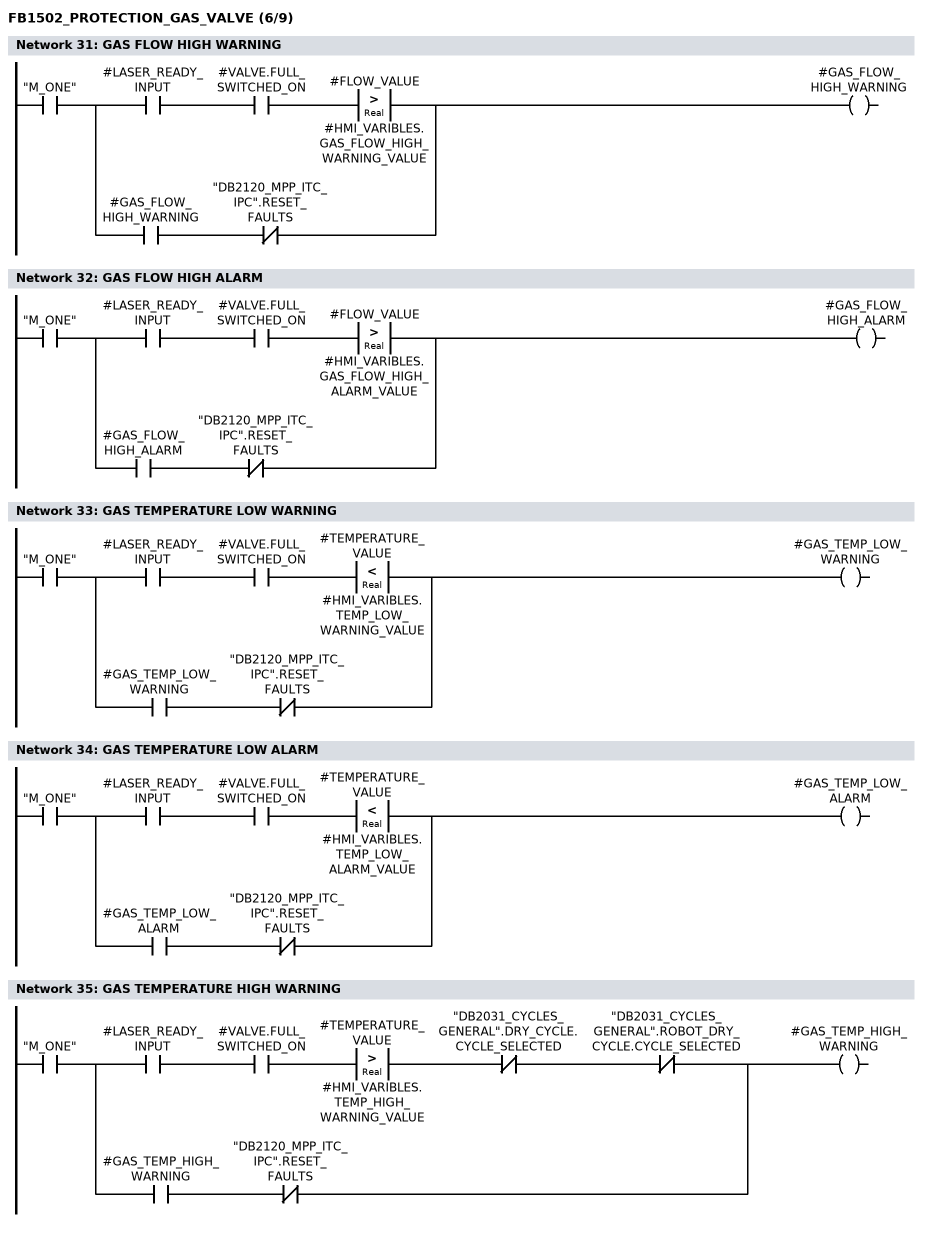
   RUNG wire#powerrail
      Contact( "M_ONE" )
      wire#w1
      Contact( #LASER_READY_INPUT )
      Contact( #VALVE.FULL_SWITCHED_ON )
      { S7_Templates := "SrcType := Real" } GT_Contact(in1 := #FLOW_VALUE, in2 := #HMI_VARIBLES.GAS_FLOW_HIGH_WARNING_VALUE)
      wire#w2
      Coil( #GAS_FLOW_HIGH_WARNING )
   END_RUNG
   RUNG wire#w1
      Contact( #GAS_FLOW_HIGH_WARNING )
      I_Contact( "DB2120_MPP_ITC_IPC".RESET_FAULTS )
   END_RUNG wire#w2
   // the same network as SCL:
   #GAS_FLOW_HIGH_WARNING := "M_ONE" AND ((#LASER_READY_INPUT AND #VALVE.FULL_SWITCHED_ON AND (#FLOW_VALUE > #HMI_VARIBLES.GAS_FLOW_HIGH_WARNING_VALUE)) OR (#GAS_FLOW_HIGH_WARNING AND NOT "DB2120_MPP_ITC_IPC".RESET_FAULTS));
END_REGION

REGION Network 32: GAS FLOW HIGH ALARM
   RUNG wire#powerrail
      Contact( "M_ONE" )
      wire#w1
      Contact( #LASER_READY_INPUT )
      Contact( #VALVE.FULL_SWITCHED_ON )
      { S7_Templates := "SrcType := Real" } GT_Contact(in1 := #FLOW_VALUE, in2 := #HMI_VARIBLES.GAS_FLOW_HIGH_ALARM_VALUE)
      wire#w2
      Coil( #GAS_FLOW_HIGH_ALARM )
   END_RUNG
   RUNG wire#w1
      Contact( #GAS_FLOW_HIGH_ALARM )
      I_Contact( "DB2120_MPP_ITC_IPC".RESET_FAULTS )
   END_RUNG wire#w2
   // the same network as SCL:
   #GAS_FLOW_HIGH_ALARM := "M_ONE" AND ((#LASER_READY_INPUT AND #VALVE.FULL_SWITCHED_ON AND (#FLOW_VALUE > #HMI_VARIBLES.GAS_FLOW_HIGH_ALARM_VALUE)) OR (#GAS_FLOW_HIGH_ALARM AND NOT "DB2120_MPP_ITC_IPC".RESET_FAULTS));
END_REGION

REGION Network 33: GAS TEMPERATURE LOW WARNING
   RUNG wire#powerrail
      Contact( "M_ONE" )
      wire#w1
      Contact( #LASER_READY_INPUT )
      Contact( #VALVE.FULL_SWITCHED_ON )
      { S7_Templates := "SrcType := Real" } LT_Contact(in1 := #TEMPERATURE_VALUE, in2 := #HMI_VARIBLES.TEMP_LOW_WARNING_VALUE)
      wire#w2
      Coil( #GAS_TEMP_LOW_WARNING )
   END_RUNG
   RUNG wire#w1
      Contact( #GAS_TEMP_LOW_WARNING )
      I_Contact( "DB2120_MPP_ITC_IPC".RESET_FAULTS )
   END_RUNG wire#w2
   // the same network as SCL:
   #GAS_TEMP_LOW_WARNING := "M_ONE" AND ((#LASER_READY_INPUT AND #VALVE.FULL_SWITCHED_ON AND (#TEMPERATURE_VALUE < #HMI_VARIBLES.TEMP_LOW_WARNING_VALUE)) OR (#GAS_TEMP_LOW_WARNING AND NOT "DB2120_MPP_ITC_IPC".RESET_FAULTS));
END_REGION

REGION Network 34: GAS TEMPERATURE LOW ALARM
   RUNG wire#powerrail
      Contact( "M_ONE" )
      wire#w1
      Contact( #LASER_READY_INPUT )
      Contact( #VALVE.FULL_SWITCHED_ON )
      { S7_Templates := "SrcType := Real" } LT_Contact(in1 := #TEMPERATURE_VALUE, in2 := #HMI_VARIBLES.TEMP_LOW_ALARM_VALUE)
      wire#w2
      Coil( #GAS_TEMP_LOW_ALARM )
   END_RUNG
   RUNG wire#w1
      Contact( #GAS_TEMP_LOW_ALARM )
      I_Contact( "DB2120_MPP_ITC_IPC".RESET_FAULTS )
   END_RUNG wire#w2
   // the same network as SCL:
   #GAS_TEMP_LOW_ALARM := "M_ONE" AND ((#LASER_READY_INPUT AND #VALVE.FULL_SWITCHED_ON AND (#TEMPERATURE_VALUE < #HMI_VARIBLES.TEMP_LOW_ALARM_VALUE)) OR (#GAS_TEMP_LOW_ALARM AND NOT "DB2120_MPP_ITC_IPC".RESET_FAULTS));
END_REGION

REGION Network 35: GAS TEMPERATURE HIGH WARNING
   RUNG wire#powerrail
      Contact( "M_ONE" )
      wire#w1
      Contact( #LASER_READY_INPUT )
      Contact( #VALVE.FULL_SWITCHED_ON )
      { S7_Templates := "SrcType := Real" } GT_Contact(in1 := #TEMPERATURE_VALUE, in2 := #HMI_VARIBLES.TEMP_HIGH_WARNING_VALUE)
      I_Contact( "DB2031_CYCLES_GENERAL".DRY_CYCLE.CYCLE_SELECTED )
      I_Contact( "DB2031_CYCLES_GENERAL".ROBOT_DRY_CYCLE.CYCLE_SELECTED )
      wire#w2
      Coil( #GAS_TEMP_HIGH_WARNING )
   END_RUNG
   RUNG wire#w1
      Contact( #GAS_TEMP_HIGH_WARNING )
      I_Contact( "DB2120_MPP_ITC_IPC".RESET_FAULTS )
   END_RUNG wire#w2
   // the same network as SCL:
   #GAS_TEMP_HIGH_WARNING := "M_ONE" AND ((#LASER_READY_INPUT AND #VALVE.FULL_SWITCHED_ON AND (#TEMPERATURE_VALUE > #HMI_VARIBLES.TEMP_HIGH_WARNING_VALUE) AND NOT "DB2031_CYCLES_GENERAL".DRY_CYCLE.CYCLE_SELECTED AND NOT "DB2031_CYCLES_GENERAL".ROBOT_DRY_CYCLE.CYCLE_SELECTED) OR (#GAS_TEMP_HIGH_WARNING AND NOT "DB2120_MPP_ITC_IPC".RESET_FAULTS));
END_REGION

REGION Network 36: GAS TEMPERATURE HIGH ALARM
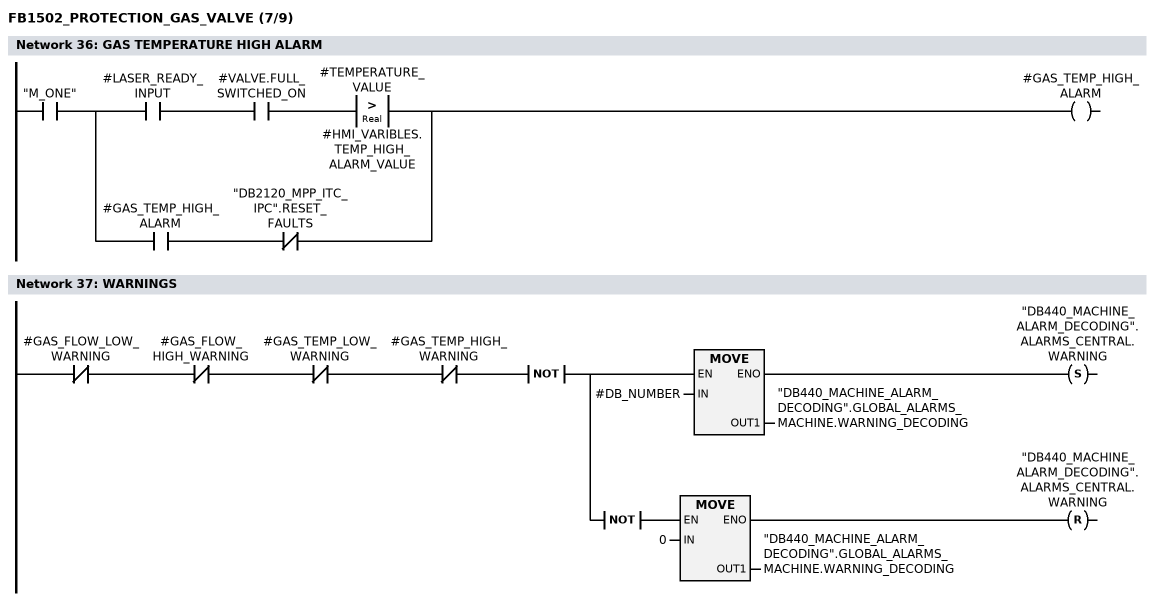
   RUNG wire#powerrail
      Contact( "M_ONE" )
      wire#w1
      Contact( #LASER_READY_INPUT )
      Contact( #VALVE.FULL_SWITCHED_ON )
      { S7_Templates := "SrcType := Real" } GT_Contact(in1 := #TEMPERATURE_VALUE, in2 := #HMI_VARIBLES.TEMP_HIGH_ALARM_VALUE)
      wire#w2
      Coil( #GAS_TEMP_HIGH_ALARM )
   END_RUNG
   RUNG wire#w1
      Contact( #GAS_TEMP_HIGH_ALARM )
      I_Contact( "DB2120_MPP_ITC_IPC".RESET_FAULTS )
   END_RUNG wire#w2
   // the same network as SCL:
   #GAS_TEMP_HIGH_ALARM := "M_ONE" AND ((#LASER_READY_INPUT AND #VALVE.FULL_SWITCHED_ON AND (#TEMPERATURE_VALUE > #HMI_VARIBLES.TEMP_HIGH_ALARM_VALUE)) OR (#GAS_TEMP_HIGH_ALARM AND NOT "DB2120_MPP_ITC_IPC".RESET_FAULTS));
END_REGION

REGION Network 37: WARNINGS
   RUNG wire#powerrail
      I_Contact( #GAS_FLOW_LOW_WARNING )
      I_Contact( #GAS_FLOW_HIGH_WARNING )
      I_Contact( #GAS_TEMP_LOW_WARNING )
      I_Contact( #GAS_TEMP_HIGH_WARNING )
      Not()
      wire#w1
      Move(in := #DB_NUMBER, out1 => "DB440_MACHINE_ALARM_DECODING".GLOBAL_ALARMS_MACHINE.WARNING_DECODING)
      S_Coil( "DB440_MACHINE_ALARM_DECODING".ALARMS_CENTRAL.WARNING )
   END_RUNG
   RUNG wire#w1
      Not()
      Move(in := 0, out1 => "DB440_MACHINE_ALARM_DECODING".GLOBAL_ALARMS_MACHINE.WARNING_DECODING)
      R_Coil( "DB440_MACHINE_ALARM_DECODING".ALARMS_CENTRAL.WARNING )
   END_RUNG
   // the same network as SCL:
   #_w1 := NOT (NOT #GAS_FLOW_LOW_WARNING AND NOT #GAS_FLOW_HIGH_WARNING AND NOT #GAS_TEMP_LOW_WARNING AND NOT #GAS_TEMP_HIGH_WARNING);
   IF #_w1 THEN
       "DB440_MACHINE_ALARM_DECODING".GLOBAL_ALARMS_MACHINE.WARNING_DECODING := #DB_NUMBER;
       "DB440_MACHINE_ALARM_DECODING".ALARMS_CENTRAL.WARNING := TRUE;
   END_IF;
   IF NOT #_w1 THEN
       "DB440_MACHINE_ALARM_DECODING".GLOBAL_ALARMS_MACHINE.WARNING_DECODING := 0;
       "DB440_MACHINE_ALARM_DECODING".ALARMS_CENTRAL.WARNING := FALSE;
   END_IF;
END_REGION

REGION Network 38: IMMEDIATE STOP AND STOP END OF CYCLE ALARMS / ALARMS CLOSED/OPENED
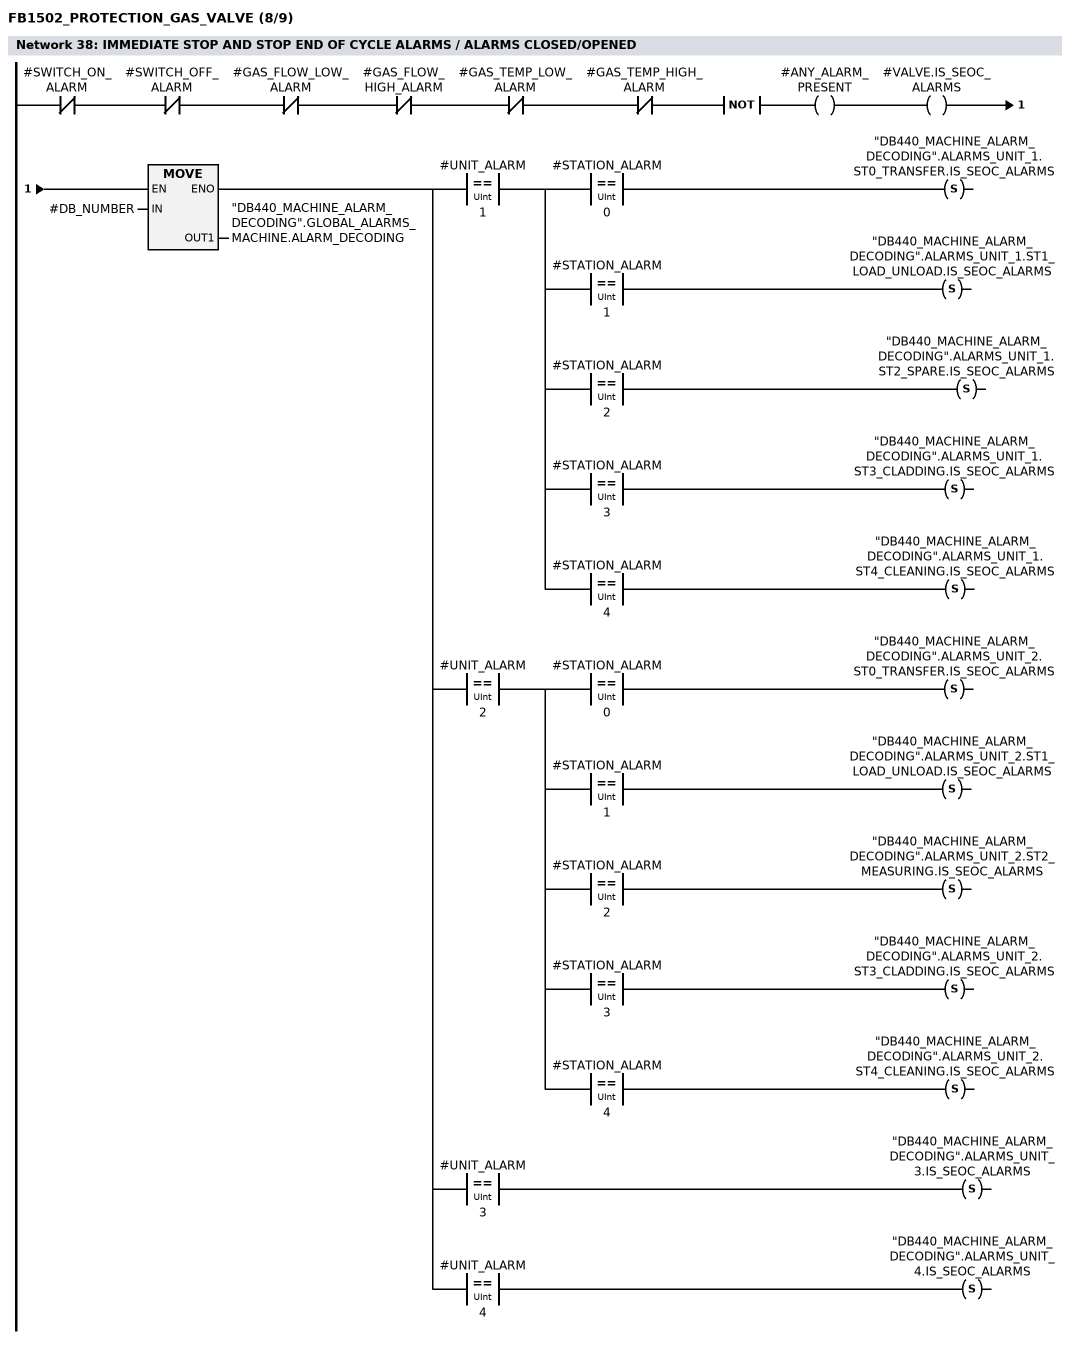
   RUNG wire#powerrail
      I_Contact( #SWITCH_ON_ALARM )
      I_Contact( #SWITCH_OFF_ALARM )
      I_Contact( #GAS_FLOW_LOW_ALARM )
      I_Contact( #GAS_FLOW_HIGH_ALARM )
      I_Contact( #GAS_TEMP_LOW_ALARM )
      I_Contact( #GAS_TEMP_HIGH_ALARM )
      Not()
      Coil( #ANY_ALARM_PRESENT )
      Coil( #VALVE.IS_SEOC_ALARMS )
      { S7_GenerateENO := "TRUE" } Move(in := #DB_NUMBER, out1 => "DB440_MACHINE_ALARM_DECODING".GLOBAL_ALARMS_MACHINE.ALARM_DECODING)
      wire#w1
      { S7_Templates := "SrcType := UInt" } EQ_Contact(in1 := #UNIT_ALARM, in2 := 1)
      wire#w2
      { S7_Templates := "SrcType := UInt" } EQ_Contact(in1 := #STATION_ALARM, in2 := 0)
      S_Coil( "DB440_MACHINE_ALARM_DECODING".ALARMS_UNIT_1.ST0_TRANSFER.IS_SEOC_ALARMS )
   END_RUNG
   RUNG wire#w2
      { S7_Templates := "SrcType := UInt" } EQ_Contact(in1 := #STATION_ALARM, in2 := 1)
      S_Coil( "DB440_MACHINE_ALARM_DECODING".ALARMS_UNIT_1.ST1_LOAD_UNLOAD.IS_SEOC_ALARMS )
   END_RUNG
   RUNG wire#w2
      { S7_Templates := "SrcType := UInt" } EQ_Contact(in1 := #STATION_ALARM, in2 := 2)
      S_Coil( "DB440_MACHINE_ALARM_DECODING".ALARMS_UNIT_1.ST2_SPARE.IS_SEOC_ALARMS )
   END_RUNG
   RUNG wire#w2
      { S7_Templates := "SrcType := UInt" } EQ_Contact(in1 := #STATION_ALARM, in2 := 3)
      S_Coil( "DB440_MACHINE_ALARM_DECODING".ALARMS_UNIT_1.ST3_CLADDING.IS_SEOC_ALARMS )
   END_RUNG
   RUNG wire#w2
      { S7_Templates := "SrcType := UInt" } EQ_Contact(in1 := #STATION_ALARM, in2 := 4)
      S_Coil( "DB440_MACHINE_ALARM_DECODING".ALARMS_UNIT_1.ST4_CLEANING.IS_SEOC_ALARMS )
   END_RUNG
   RUNG wire#w1
      { S7_Templates := "SrcType := UInt" } EQ_Contact(in1 := #UNIT_ALARM, in2 := 2)
      wire#w3
      { S7_Templates := "SrcType := UInt" } EQ_Contact(in1 := #STATION_ALARM, in2 := 0)
      S_Coil( "DB440_MACHINE_ALARM_DECODING".ALARMS_UNIT_2.ST0_TRANSFER.IS_SEOC_ALARMS )
   END_RUNG
   RUNG wire#w3
      { S7_Templates := "SrcType := UInt" } EQ_Contact(in1 := #STATION_ALARM, in2 := 1)
      S_Coil( "DB440_MACHINE_ALARM_DECODING".ALARMS_UNIT_2.ST1_LOAD_UNLOAD.IS_SEOC_ALARMS )
   END_RUNG
   RUNG wire#w3
      { S7_Templates := "SrcType := UInt" } EQ_Contact(in1 := #STATION_ALARM, in2 := 2)
      S_Coil( "DB440_MACHINE_ALARM_DECODING".ALARMS_UNIT_2.ST2_MEASURING.IS_SEOC_ALARMS )
   END_RUNG
   RUNG wire#w3
      { S7_Templates := "SrcType := UInt" } EQ_Contact(in1 := #STATION_ALARM, in2 := 3)
      S_Coil( "DB440_MACHINE_ALARM_DECODING".ALARMS_UNIT_2.ST3_CLADDING.IS_SEOC_ALARMS )
   END_RUNG
   RUNG wire#w3
      { S7_Templates := "SrcType := UInt" } EQ_Contact(in1 := #STATION_ALARM, in2 := 4)
      S_Coil( "DB440_MACHINE_ALARM_DECODING".ALARMS_UNIT_2.ST4_CLEANING.IS_SEOC_ALARMS )
   END_RUNG
   RUNG wire#w1
      { S7_Templates := "SrcType := UInt" } EQ_Contact(in1 := #UNIT_ALARM, in2 := 3)
      S_Coil( "DB440_MACHINE_ALARM_DECODING".ALARMS_UNIT_3.IS_SEOC_ALARMS )
   END_RUNG
   RUNG wire#w1
      { S7_Templates := "SrcType := UInt" } EQ_Contact(in1 := #UNIT_ALARM, in2 := 4)
      S_Coil( "DB440_MACHINE_ALARM_DECODING".ALARMS_UNIT_4.IS_SEOC_ALARMS )
   END_RUNG
   // the same network as SCL:
   // ENO of a box is taken as its EN; it also drops when the box reports an error
   #ANY_ALARM_PRESENT := NOT (NOT #SWITCH_ON_ALARM AND NOT #SWITCH_OFF_ALARM AND NOT #GAS_FLOW_LOW_ALARM AND NOT #GAS_FLOW_HIGH_ALARM AND NOT #GAS_TEMP_LOW_ALARM AND NOT #GAS_TEMP_HIGH_ALARM);
   #VALVE.IS_SEOC_ALARMS := #ANY_ALARM_PRESENT;
   IF #ANY_ALARM_PRESENT THEN
       "DB440_MACHINE_ALARM_DECODING".GLOBAL_ALARMS_MACHINE.ALARM_DECODING := #DB_NUMBER;
   END_IF;
   #_w1 := #ANY_ALARM_PRESENT AND (#UNIT_ALARM = 1);
   IF #_w1 AND (#STATION_ALARM = 0) THEN
       "DB440_MACHINE_ALARM_DECODING".ALARMS_UNIT_1.ST0_TRANSFER.IS_SEOC_ALARMS := TRUE;
   END_IF;
   IF #_w1 AND (#STATION_ALARM = 1) THEN
       "DB440_MACHINE_ALARM_DECODING".ALARMS_UNIT_1.ST1_LOAD_UNLOAD.IS_SEOC_ALARMS := TRUE;
   END_IF;
   IF #_w1 AND (#STATION_ALARM = 2) THEN
       "DB440_MACHINE_ALARM_DECODING".ALARMS_UNIT_1.ST2_SPARE.IS_SEOC_ALARMS := TRUE;
   END_IF;
   IF #_w1 AND (#STATION_ALARM = 3) THEN
       "DB440_MACHINE_ALARM_DECODING".ALARMS_UNIT_1.ST3_CLADDING.IS_SEOC_ALARMS := TRUE;
   END_IF;
   IF #_w1 AND (#STATION_ALARM = 4) THEN
       "DB440_MACHINE_ALARM_DECODING".ALARMS_UNIT_1.ST4_CLEANING.IS_SEOC_ALARMS := TRUE;
   END_IF;
   #_w2 := #ANY_ALARM_PRESENT AND (#UNIT_ALARM = 2);
   IF #_w2 AND (#STATION_ALARM = 0) THEN
       "DB440_MACHINE_ALARM_DECODING".ALARMS_UNIT_2.ST0_TRANSFER.IS_SEOC_ALARMS := TRUE;
   END_IF;
   IF #_w2 AND (#STATION_ALARM = 1) THEN
       "DB440_MACHINE_ALARM_DECODING".ALARMS_UNIT_2.ST1_LOAD_UNLOAD.IS_SEOC_ALARMS := TRUE;
   END_IF;
   IF #_w2 AND (#STATION_ALARM = 2) THEN
       "DB440_MACHINE_ALARM_DECODING".ALARMS_UNIT_2.ST2_MEASURING.IS_SEOC_ALARMS := TRUE;
   END_IF;
   IF #_w2 AND (#STATION_ALARM = 3) THEN
       "DB440_MACHINE_ALARM_DECODING".ALARMS_UNIT_2.ST3_CLADDING.IS_SEOC_ALARMS := TRUE;
   END_IF;
   IF #_w2 AND (#STATION_ALARM = 4) THEN
       "DB440_MACHINE_ALARM_DECODING".ALARMS_UNIT_2.ST4_CLEANING.IS_SEOC_ALARMS := TRUE;
   END_IF;
   IF #ANY_ALARM_PRESENT AND (#UNIT_ALARM = 3) THEN
       "DB440_MACHINE_ALARM_DECODING".ALARMS_UNIT_3.IS_SEOC_ALARMS := TRUE;
   END_IF;
   IF #ANY_ALARM_PRESENT AND (#UNIT_ALARM = 4) THEN
       "DB440_MACHINE_ALARM_DECODING".ALARMS_UNIT_4.IS_SEOC_ALARMS := TRUE;
   END_IF;
END_REGION

REGION Network 39: ANY ACTIVE ALARM
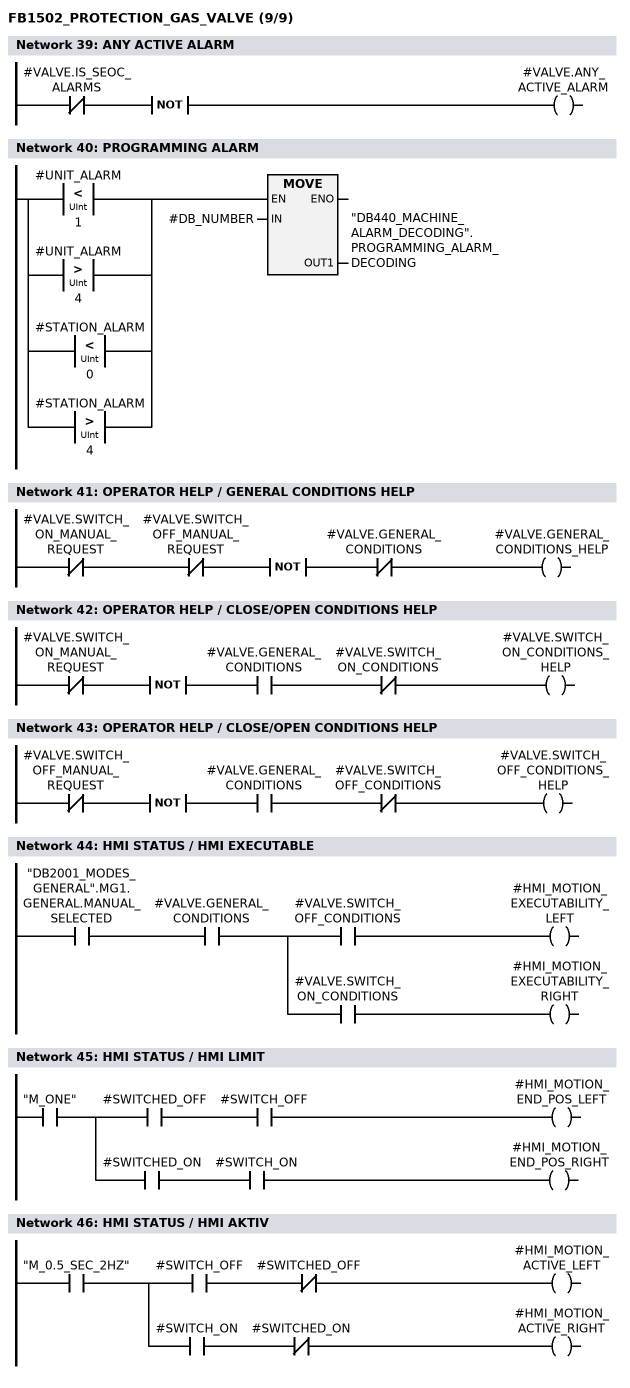
   RUNG wire#powerrail
      I_Contact( #VALVE.IS_SEOC_ALARMS )
      Not()
      Coil( #VALVE.ANY_ACTIVE_ALARM )
   END_RUNG
   // the same network as SCL:
   #VALVE.ANY_ACTIVE_ALARM := NOT (NOT #VALVE.IS_SEOC_ALARMS);
END_REGION

REGION Network 40: PROGRAMMING ALARM
   RUNG wire#powerrail
      { S7_Templates := "SrcType := UInt" } LT_Contact(in1 := #UNIT_ALARM, in2 := 1)
      wire#w1
      Move(in := #DB_NUMBER, out1 => "DB440_MACHINE_ALARM_DECODING".PROGRAMMING_ALARM_DECODING)
   END_RUNG
   RUNG wire#powerrail
      { S7_Templates := "SrcType := UInt" } GT_Contact(in1 := #UNIT_ALARM, in2 := 4)
   END_RUNG wire#w1
   RUNG wire#powerrail
      { S7_Templates := "SrcType := UInt" } LT_Contact(in1 := #STATION_ALARM, in2 := 0)
   END_RUNG wire#w1
   RUNG wire#powerrail
      { S7_Templates := "SrcType := UInt" } GT_Contact(in1 := #STATION_ALARM, in2 := 4)
   END_RUNG wire#w1
   // the same network as SCL:
   IF (#UNIT_ALARM < 1) OR (#UNIT_ALARM > 4) OR (#STATION_ALARM < 0) OR (#STATION_ALARM > 4) THEN
       "DB440_MACHINE_ALARM_DECODING".PROGRAMMING_ALARM_DECODING := #DB_NUMBER;
   END_IF;
END_REGION

REGION Network 41: OPERATOR HELP / GENERAL CONDITIONS HELP
   RUNG wire#powerrail
      I_Contact( #VALVE.SWITCH_ON_MANUAL_REQUEST )
      I_Contact( #VALVE.SWITCH_OFF_MANUAL_REQUEST )
      Not()
      I_Contact( #VALVE.GENERAL_CONDITIONS )
      Coil( #VALVE.GENERAL_CONDITIONS_HELP )
   END_RUNG
   // the same network as SCL:
   #VALVE.GENERAL_CONDITIONS_HELP := NOT (NOT #VALVE.SWITCH_ON_MANUAL_REQUEST AND NOT #VALVE.SWITCH_OFF_MANUAL_REQUEST) AND NOT #VALVE.GENERAL_CONDITIONS;
END_REGION

REGION Network 42: OPERATOR HELP / CLOSE/OPEN CONDITIONS HELP
   RUNG wire#powerrail
      I_Contact( #VALVE.SWITCH_ON_MANUAL_REQUEST )
      Not()
      Contact( #VALVE.GENERAL_CONDITIONS )
      I_Contact( #VALVE.SWITCH_ON_CONDITIONS )
      Coil( #VALVE.SWITCH_ON_CONDITIONS_HELP )
   END_RUNG
   // the same network as SCL:
   #VALVE.SWITCH_ON_CONDITIONS_HELP := NOT (NOT #VALVE.SWITCH_ON_MANUAL_REQUEST) AND #VALVE.GENERAL_CONDITIONS AND NOT #VALVE.SWITCH_ON_CONDITIONS;
END_REGION

REGION Network 43: OPERATOR HELP / CLOSE/OPEN CONDITIONS HELP
   RUNG wire#powerrail
      I_Contact( #VALVE.SWITCH_OFF_MANUAL_REQUEST )
      Not()
      Contact( #VALVE.GENERAL_CONDITIONS )
      I_Contact( #VALVE.SWITCH_OFF_CONDITIONS )
      Coil( #VALVE.SWITCH_OFF_CONDITIONS_HELP )
   END_RUNG
   // the same network as SCL:
   #VALVE.SWITCH_OFF_CONDITIONS_HELP := NOT (NOT #VALVE.SWITCH_OFF_MANUAL_REQUEST) AND #VALVE.GENERAL_CONDITIONS AND NOT #VALVE.SWITCH_OFF_CONDITIONS;
END_REGION

REGION Network 44: HMI STATUS / HMI EXECUTABLE
   RUNG wire#powerrail
      Contact( "DB2001_MODES_GENERAL".MG1.GENERAL.MANUAL_SELECTED )
      Contact( #VALVE.GENERAL_CONDITIONS )
      wire#w1
      Contact( #VALVE.SWITCH_OFF_CONDITIONS )
      Coil( #HMI_MOTION_EXECUTABILITY_LEFT )
   END_RUNG
   RUNG wire#w1
      Contact( #VALVE.SWITCH_ON_CONDITIONS )
      Coil( #HMI_MOTION_EXECUTABILITY_RIGHT )
   END_RUNG
   // the same network as SCL:
   #_w1 := "DB2001_MODES_GENERAL".MG1.GENERAL.MANUAL_SELECTED AND #VALVE.GENERAL_CONDITIONS;
   #HMI_MOTION_EXECUTABILITY_LEFT := #_w1 AND #VALVE.SWITCH_OFF_CONDITIONS;
   #HMI_MOTION_EXECUTABILITY_RIGHT := #_w1 AND #VALVE.SWITCH_ON_CONDITIONS;
END_REGION

REGION Network 45: HMI STATUS / HMI LIMIT
   RUNG wire#powerrail
      Contact( "M_ONE" )
      wire#w1
      Contact( #SWITCHED_OFF )
      Contact( #SWITCH_OFF )
      Coil( #HMI_MOTION_END_POS_LEFT )
   END_RUNG
   RUNG wire#w1
      Contact( #SWITCHED_ON )
      Contact( #SWITCH_ON )
      Coil( #HMI_MOTION_END_POS_RIGHT )
   END_RUNG
   // the same network as SCL:
   #HMI_MOTION_END_POS_LEFT := "M_ONE" AND #SWITCHED_OFF AND #SWITCH_OFF;
   #HMI_MOTION_END_POS_RIGHT := "M_ONE" AND #SWITCHED_ON AND #SWITCH_ON;
END_REGION

REGION Network 46: HMI STATUS / HMI AKTIV
   RUNG wire#powerrail
      Contact( "M_0.5_SEC_2HZ" )
      wire#w1
      Contact( #SWITCH_OFF )
      I_Contact( #SWITCHED_OFF )
      Coil( #HMI_MOTION_ACTIVE_LEFT )
   END_RUNG
   RUNG wire#w1
      Contact( #SWITCH_ON )
      I_Contact( #SWITCHED_ON )
      Coil( #HMI_MOTION_ACTIVE_RIGHT )
   END_RUNG
   // the same network as SCL:
   #HMI_MOTION_ACTIVE_LEFT := "M_0.5_SEC_2HZ" AND #SWITCH_OFF AND NOT #SWITCHED_OFF;
   #HMI_MOTION_ACTIVE_RIGHT := "M_0.5_SEC_2HZ" AND #SWITCH_ON AND NOT #SWITCHED_ON;
END_REGION
END_FUNCTION_BLOCK
